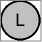
VISUALIZATION V_Licht  // 42x42
VAR_IN_OUT
	m_Input_fbLicht : FB_Licht;
END_VAR
    Ellipse (0,0 40x40), "L", colour toggle: (m_Input_fbLicht.QbOutLicht) <> 0
        tap m_Input_fbLicht.bInVisu
    Polyline (30,30)
    Polyline (0,0)
    Polyline (30,10)
    Polyline (10,30)
END_VISUALIZATION

(* stored: Version 1.1.0.1, ProductVersion 3.1.4018.5
   Visu V_Licht: Id {cc93e8b3-4598-4ce3-9b18-7697775f2dc2} *)
